# EPICS autosave request: iocs/eigerIOC/iocBoot/iocEiger2/auto_settings.req
file "eiger_settings.req",        P=$(P),  R=cam1:
file "NDStdArrays_settings.req",  P=$(P),  R=image1:
file "NDStdArrays_settings.req",  P=$(P),  R=image2:
file "commonPlugin_settings.req", P=$(P)
